{attribute 'pack_mode' := '2'}
TYPE ST_XTS_TRANSPORT_CTRL :
STRUCT
  Cmd       : E_XTS_TRANSPORT_CTRL;
END_STRUCT
END_TYPE

(* stored: Version 1.1.0.1
   DUT ST_XTS_TRANSPORT_CTRL: Id {cc0196e2-81cc-4d95-82b0-a196b1e47936} *)
